FUNCTION IsInRangeInclusive3D : BOOL
VAR_INPUT
	point : Point3D;
	range : Range3D;
END_VAR

IsInRangeInclusive3D := 
	IsInRangeInclusive(point.X, range.X)
	AND IsInRangeInclusive(point.Y, range.Y)
	AND IsInRangeInclusive(point.Z, range.Z)
	;

END_FUNCTION

(* stored: Version 1.1.0.1, ProductVersion 3.1.4024.15
   POU IsInRangeInclusive3D: Id {a7196623-68ee-0cc8-2adb-437e06286091}, SpecialFunc None *)
